// TIA Portal V20 export
TYPE "typeEm6MonitoringCmStatus"
// stored: Access Published, Namespace Unit1
   STRUCT
      visionAixs { ExternalWritable := 'False'} : "LBC_typeAxis64PosControlNodeMonitoring";
      visionPusherSupport { ExternalWritable := 'False'} : "LBC_typeTwoWayActuatorControlNodeMonitoring";
      visionTriggerSensor { ExternalWritable := 'False'} : "LBC_typeDigitalSignalControlNodeMonitoring";
      visionController { ExternalWritable := 'False'} : "LER_typeVisionMonitoring";
   END_STRUCT;
END_TYPE
